FUNCTION_BLOCK INTERNAL StringBuilder IMPLEMENTS IStringBuilder, ILimitedStringBuilder
VAR
  {attribute 'hide'}
  _workString : Tc2_System.T_MaxString;
END_VAR

METHOD PUBLIC Append : IStringBuilder // Append text TO t current build STRING.
VAR_INPUT
  text : Tc2_System.T_MaxString; //text to append to current build string
END_VAR
_workString:= Tc2_Standard.CONCAT(_workString,text);
Append := THIS^;
END_METHOD

METHOD PUBLIC AppendIf : IStringBuilder
VAR_INPUT
  condition : BOOL;
  text : Tc2_System.T_MaxString;
END_VAR
IF condition THEN
  _workString:= Tc2_Standard.CONCAT(_workString,text);
END_IF
AppendIf := THIS^;
END_METHOD

METHOD PUBLIC InsertAtLocation : IStringBuilder
VAR_INPUT
  text : Tc2_System.T_MaxString;
  position : INT;
END_VAR
_workString := Tc2_Standard.INSERT(_workSTring,text,position);
InsertAtLocation  := THIS^;
END_METHOD

METHOD PadLeft : IStringBuilder
VAR_INPUT
  text : Tc2_System.T_MaxString; // Text to append to current build string
  length : INT; // Total length of text + padding
  c : STRING(1); // Character to be padded left of text
END_VAR
VAR
  i : INT;
  padLength : INT;
END_VAR
// Add left padding
padLength := Tc2_Standard.LEN(text) - length;
FOR i := 1 TO padLength DO
  _workString:= Tc2_Standard.CONCAT(_workString, c);
END_FOR

// Add text
_workString:= Tc2_Standard.CONCAT(_workString,text);

PadLeft := THIS^;
END_METHOD

METHOD PUBLIC Reset : ILimitedStringBuilder //Reset current build STRING TO an empty STRING.
_workString:='';
Reset := THIS^;
END_METHOD

METHOD PUBLIC ToString : Tc2_System.T_MaxString //Returns current build STRING.
ToString := _workString;
END_METHOD

END_FUNCTION_BLOCK

(* stored: Version 1.1.0.1
   POU StringBuilder: Id {368e5049-935b-4562-a874-cb9be5225f7d}, SpecialFunc None
   Method Append: Id {3f45997e-6006-457f-9a9a-30ac281e8f8a}
   Method AppendIf: Id {341a7b9c-f058-4735-b313-3a46f602e9e1}
   Method InsertAtLocation: Id {b2ed9ced-aca1-4991-af8e-c808997da606}
   Method PadLeft: Id {26c6478b-ece5-418e-9b19-10604dda05cb}
   Method Reset: Id {f04f2676-7659-44a8-87c7-48fdd5328c04}
   Method ToString: Id {8c20dc6d-f3fa-4203-b887-d1b9b96ecacc} *)
